// TIA Portal project "SortinStation" (V15)
// Vorlageprojekt für das Buch mit Zielsystem S7-1200

(* hardware
DEVICE "S7-1200-Station_1"  S7-1200 Station
   slot 0: "Baugruppenträger_0"  Rack  V1.0
   slot 1: "PLC_1"  CPU 1211C DC/DC/DC  6ES7 211-1AE40-0XB0  V4.1
*)

// ===== PLC "PLC_1"  CPU 1211C DC/DC/DC =====

VAR_GLOBAL   // PLC tag table "Standard-Variablentabelle"
   "Entry Conveyor" AT %A0.0 : Bool;
   "Tag_2" AT %E0.0 : Bool;
   "Start" AT %E0.1 : Bool;
   "Stop" AT %I0.3 : Bool;
   "Vision Sensor" AT %ID30 : DWord;
   "Tag_6" AT %I0.7 : Bool;
   "Tag_7" AT %ID31 : DWord;
   "Tag_8" AT %ID32 : DInt;
   "Tag_9" AT %Q0.3 : Bool;
   "Tag_10" AT %Q0.7 : Bool;
   "Exit Conveyor" AT %Q0.2 : Bool;
   "Sorter 2 Turn" AT %Q0.5 : Bool;
   "Timmer 2 Valve" AT %Q1.4 : Bool;
   "Sorter 1 Belt" AT %Q0.4 : Bool;
   "Sorter 2 Belt" AT %Q0.6 : Bool;
   "Sorter 3 Belt" AT %Q1.0 : Bool;
   "Tag_17" AT %Q1.5 : Bool;
   "Tag_18" AT %Q1.6 : Bool;
END_VAR

// folder: System blocks/Program resources

DATA_BLOCK "IEC_Timer_0_DB"   // DB1
{ S7_Optimized_Access := 'TRUE' }
AUTHOR : Simatic
FAMILY : IEC
NAME : IEC_TMR
VERSION : 1.0
// stored: InstanceOfName IEC_TIMER
"IEC_TIMER"
BEGIN
END_DATA_BLOCK

DATA_BLOCK "IEC_Timer_0_DB_1"   // DB2
{ S7_Optimized_Access := 'TRUE' }
AUTHOR : Simatic
FAMILY : IEC
NAME : IEC_TMR
VERSION : 1.0
// stored: InstanceOfName IEC_TIMER
"IEC_TIMER"
BEGIN
END_DATA_BLOCK

DATA_BLOCK "IEC_Timer_0_DB_2"   // DB3
{ S7_Optimized_Access := 'TRUE' }
AUTHOR : Simatic
FAMILY : IEC
NAME : IEC_TMR
VERSION : 1.0
// stored: InstanceOfName IEC_TIMER
"IEC_TIMER"
BEGIN
END_DATA_BLOCK

DATA_BLOCK "IEC_Timer_0_DB_3"   // DB4
{ S7_Optimized_Access := 'TRUE' }
AUTHOR : Simatic
FAMILY : IEC
NAME : IEC_TMR
VERSION : 1.0
// stored: InstanceOfName IEC_TIMER
"IEC_TIMER"
BEGIN
END_DATA_BLOCK

DATA_BLOCK "IEC_Timer_0_DB_4"   // DB5
{ S7_Optimized_Access := 'TRUE' }
AUTHOR : Simatic
FAMILY : IEC
NAME : IEC_TMR
VERSION : 1.0
// stored: InstanceOfName IEC_TIMER
"IEC_TIMER"
BEGIN
END_DATA_BLOCK

DATA_BLOCK "IEC_Timer_0_DB_5"   // DB6
{ S7_Optimized_Access := 'TRUE' }
AUTHOR : Simatic
FAMILY : IEC
NAME : IEC_TMR
VERSION : 1.0
// stored: InstanceOfName IEC_TIMER
"IEC_TIMER"
BEGIN
END_DATA_BLOCK

// folder: (top level)

FUNCTION "MHJ-PLC-Lab-Function-S71200" : Void   // FC9000, SCL
{ S7_Optimized_Access := 'TRUE' }
VERSION : 0.1
   VAR_TEMP
      rdTimeReturn : Int;
      outputTime : DTL;
      SyncVal : Byte;
      forVal : Int;
      forVal_2 : Int;
      Value : Byte;
   END_VAR
   VAR CONSTANT
      CompVal : Byte := 16#34;
      Value_01 : Byte := 16#11;
      Value_01_DW : DWord := 16#A165_D992;
      Value_02_DW : DWord := 16#58BE_4401;
   END_VAR
BEGIN

   #Value:=PEEK(area := 16#82,
        dbNumber := 0,
        byteOffset := 511);
   #Value := #Value + 1;

   POKE(area := 16#82,
        dbNumber := 0,
        byteOffset := 511,
        value := #Value);

   POKE(area:=16#81,
        dbNumber:=0,
        byteOffset:=1016,
        value:=#Value_01_DW);
   POKE(area := 16#81,
        dbNumber := 0,
        byteOffset := 1020,
        value := #Value_02_DW);

   POKE(area := 16#81,
        dbNumber := 0,
        byteOffset := 511,
        value := B#16#00);

   FOR #forVal := 0 TO 120 DO
       FOR #forVal_2:=0 TO 10 DO
           #rdTimeReturn:=RD_SYS_T(#outputTime);
           #rdTimeReturn := WR_SYS_T(#outputTime);
           #rdTimeReturn := RD_SYS_T(#outputTime);
           #rdTimeReturn := WR_SYS_T(#outputTime);
       END_FOR;
       #SyncVal:= PEEK(area := 16#81,
                      dbNumber := 0,
                      byteOffset := 511);
       IF #SyncVal = #CompVal THEN
          GOTO M_1;
       END_IF;
   END_FOR;
   RETURN;

   M_1:
   POKE(area := 16#81,
        dbNumber := 0,
        byteOffset := 511,
        value := B#16#0);
END_FUNCTION

ORGANIZATION_BLOCK "Main"   // OB1, LAD, ProgramCycle
TITLE = "Main Program Sweep (Cycle)"
{ S7_Optimized_Access := 'TRUE' }
VERSION : 0.1
   VAR_INPUT
      Initial_Call : Bool;   // Initial call of this OB
      Remanence : Bool;   // =True, if remanent data are available
   END_VAR
BEGIN

REGION Network 1: Konnektierungsbaustein für PLC-Lab
   // Im Netzwerk 1 wird der Konnektierungsbaustein für PLC-Lab aufgerufen.
   // Dieser Aufruf darf nicht entfernt werden!
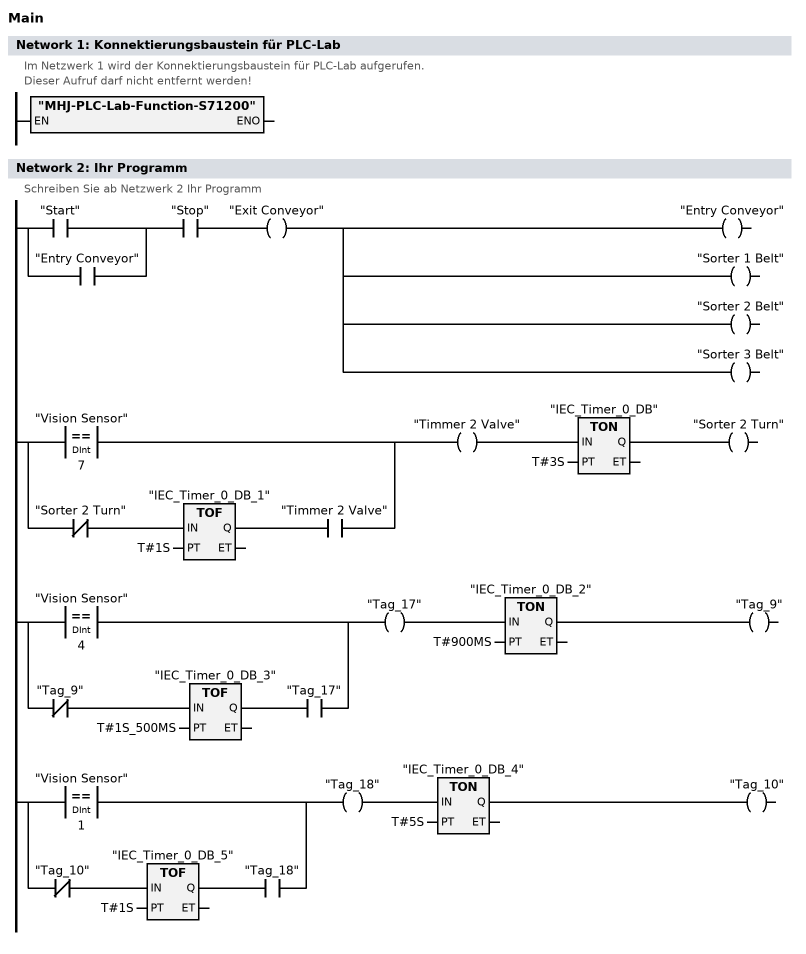
   RUNG wire#powerrail
      "MHJ-PLC-Lab-Function-S71200"()
   END_RUNG
   // the same network as SCL:
   "MHJ-PLC-Lab-Function-S71200"();
END_REGION

REGION Network 2: Ihr Programm
   // Schreiben Sie ab Netzwerk 2 Ihr Programm
   "Exit Conveyor" := ("Start" OR "Entry Conveyor") AND "Stop";
   "Entry Conveyor" := "Exit Conveyor";
   "Sorter 1 Belt" := "Exit Conveyor";
   "Sorter 2 Belt" := "Exit Conveyor";
   "Sorter 3 Belt" := "Exit Conveyor";
   "IEC_Timer_0_DB_1".TOF(IN := NOT "Sorter 2 Turn", PT := T#1S);
   "Timmer 2 Valve" := ("Vision Sensor" = 7) OR ("IEC_Timer_0_DB_1".Q AND "Timmer 2 Valve");
   "IEC_Timer_0_DB".TON(IN := "Timmer 2 Valve", PT := T#3S);
   "Sorter 2 Turn" := "IEC_Timer_0_DB".Q;
   "IEC_Timer_0_DB_3".TOF(IN := NOT "Tag_9", PT := T#1S_500MS);
   "Tag_17" := ("Vision Sensor" = 4) OR ("IEC_Timer_0_DB_3".Q AND "Tag_17");
   "IEC_Timer_0_DB_2".TON(IN := "Tag_17", PT := T#900MS);
   "Tag_9" := "IEC_Timer_0_DB_2".Q;
   "IEC_Timer_0_DB_5".TOF(IN := NOT "Tag_10", PT := T#1S);
   "Tag_18" := ("Vision Sensor" = 1) OR ("IEC_Timer_0_DB_5".Q AND "Tag_18");
   "IEC_Timer_0_DB_4".TON(IN := "Tag_18", PT := T#5S);
   "Tag_10" := "IEC_Timer_0_DB_4".Q;
END_REGION
END_ORGANIZATION_BLOCK